// SIMATIC S7-200 project (STEP 7-Micro/WIN), CPU 224 REL 01.10

SYMBOL_TABLE IN/OUT
                 I0.0     // 水流量脉冲信号 0~3HZ,对应0~540M3/h
                 I0.1     // 变频器保护
                 I0.2     // 变频器输出控制权标定 脉冲转换 PLC/人操
                 I0.3     // 1#机变频电路 应答
                 I0.4     // 1#机系统电源电路 应答
                 I0.5     // 1#机变频电路 备妥
                 I0.6     // 1#机系统电源电路 备妥
                 I0.7     // 1#机电路热保护
                 I1.0     // 音响确认/试验
                 I1.1     // 2#机变频电路 应答
                 I1.2     // 2#机系统电源电路 应答
                 I1.3     // 2#机变频电路 备妥
                 I1.4     // 2#机系统电源电路 备妥
                 I1.5     // 2#机电路热保护
                 I2.0     // 3#机系统电源电路 应答
                 I2.1     // 3#机系统电源电路 备妥
                 I2.2     // 3#机电路热保护
                 I2.3     // 备用
                 Q0.0     // 1#机(电路)变频驱动
                 Q0.1     // 1#机系统电源驱动
                 Q0.2     // 2#机(电路)变频驱动
                 Q0.3     // 2#机系统电源驱动
                 Q0.4     // 停变频 复位自启动
                 Q0.5     // 1#操作提示
                 Q0.6     // 2#操作提示
                 Q0.7     // 共同部分操作提示
                 Q1.0     // 驱动报警音响
                 Q1.1     // 变频器输出由PLC控制 驱动指示灯
                 Q2.0     // 3#机系统电源驱动
                 Q2.1     // 备用
                 Q2.2     // 备用
                 Q2.3     // 备用
                 M0.0     // F1 1#机变频电路启动/停止
                 M0.1     // F2 1#机系统电源驱动的启动/停止
                 M0.2     // F3 2#机变频电路启动/停止
                 M0.3     // F4 2#机系统电源驱动的启动/停止
                 M0.4     // F5 3#机系统电源驱动的启动/停止
                 M0.5     // F6 变频手动输出设置调出
                 M0.6     // F7 待机/手动/自动切换
                 M0.7     // F8 赋值操作调出
                 AIW0     // 给水压力
                 AIW2     // 备用
                 AIW4     // 备用
                 AIW6     // 备用
                 AQW0     // 变频器输出频率控制
                 AQW2     // 备用
END_SYMBOL_TABLE

SYMBOL_TABLE OTHER
                 VD844    // Process Variable
                 VD848    // Loop Setpoint
                 VD852    // Calculated Loop Output
                 VD856    // Loop Gain
                 VD860    // Sample Time
                 VD864    // Integral Time
                 VD1012   // 供水安全值
                 VD1016   // 泵出口压力额定值
                 VD1020   // 泵供水量额定值
END_SYMBOL_TABLE

ORGANIZATION_BLOCK MAIN:OB1
TITLE= 
// 项目、设备信息
// 供水系统由2台55kw电机驱动的离心式水泵和1台30kw水泵组成工艺设备，其中55kw电机驱动的为主供水泵，额定压头420Kpa,额定流量250M3/h。正常供水量在额定流量范围内，一开一备。30kw电机驱动的为紧急泵，特殊工况下使用。系统设计为１台主供水泵由55kw变频器驱动，实现最佳节能控制，这台变频器还用于软启动两台水泵。（通过电气切换，在１台泵变频启动后，实行变频供电和系统电源切换，转由系统电源供电，变频器再去启动另１台泵。）在某些工况下，可能２台55kw泵同时运行。系统运行方式设计为"人操"和"ＰＬＣ"两种方式。
// 
// 系统注释
// 1、系统启动时，首先通过INIT子程序将系统运行模式置为待机状态，并初始化TD200显示屏参数。
// 2、系统中，两台55kW水泵分别由水泵1变频控制输出和水泵2变频控制输出控制，通过一台55kW变频器实现软启动和变频调速，以适应用水量变化。
// 3.、通过电气切换，在1#泵变频启动后，实行变频供电和系统电源切换，转由系统电源供电，变频器再去启动2#泵。
// 4、同时，30kW的水泵3控制输出在主泵异常时作为紧急备用，由F5键控制启停。
// 5.、小区物业管理人员可以通过TD200显示屏实时查看水泵状态、压力和流量数据。
// 6.、正常运行中，程序利用流量定时器计算每台水泵的流量，存储在流量计算结果中。
// 7、同时通过压力显示定时器定期更新压力数据到显示屏，确保物业人员随时掌握供水情况。
// 8、系统支持手动和自动两种模式切换，通过F7键触发，修改模式时确保水泵1变频控制输出已稳定，避免操作冲突。
// 9、在手动模式下，操作员可通过F1键启动1#机变频运行，但需变频器无故障且就绪时才会置位。
// 10、此外，F3键和F5键分别控制2#机和3#机的启停。
// 11、变频器的频率调整通过F6键实现，输出频率被严格限制在0-50Hz范围内，以保护设备不过载。
// 12、当切换至自动模式时，系统依靠PID调节自动控制水泵运行，维持恒定水压，此功能仅在自动模式下生效。
// 13、系统还会实时监控水泵1运行反馈等信号，并在TD200上显示状态。
// 14、安全性方面，若检测到水泵1热保护故障，程序立即复位水泵1变频控制输出和系统电源输出，并通过报警音响输出发出提示。
// 15、正常情况下，TD200显示屏显示PLC及1#机泵、2#机泵、3#机泵和变频器的运行状态，以及压力和流量测量值。
// 16、当有故障发生时，TD200显示屏显示汉字报警信息，PLC驱动音响报警，并自动停止故障设备。
// 17、操作人员可按确认键确认报警信息，按音响试验/消除按钮关闭音响，然后处理故障。
// 
// 
// 附加信息
// 正常情况下，TD200显示屏显示ＰＬＣ，１＃机泵，２＃机泵，３＃机泵和变频器的运行状态以及压力和流量测量值。当有故障发生时，TD200显示屏显示汉字的报警信息，同时ＰＬＣ驱动音响进行声音报警，ＰＬＣ自动停止发生故障的电气设备，以确保安全。操作人员可按确认键确认汉字的报警信息，按音响试验／消除按钮关闭音响，然后对故障进行处理。
// 
// 
BEGIN
Network 1 // 初始化
//  
// NETWORK COMMENTS
//  
// 
LD     SM0.1
CALL   INIT:SBR0
?000
Network 2 // 使能PID控制中断程序
// 
// 
LD     SM0.0
CALL   SBR_PID:SBR8
Network 3 // 流量脉冲计时
// 
// 
LD     SM0.0
TONR   T1, +32760
Network 4
LD     SM0.0
A      T1
MOVR   0.0, VD318
AENO
MOVR   0.0, VD338
AENO
MOVR   0.0, VD358
Network 5 // 显示压力
// 
// 
LD     SM0.0
AN     M3.1
TON    T103, +10
Network 6
// 
// 
LD     SM0.0
A      T103
CALL   P_DISPLAY:SBR1
=      M3.1
Network 7 // 显示电机与变频状态
// 
// 
LD     SM0.0
CALL   S_DISPLY:SBR2
Network 8
LD     SM0.0
AN     M2.1
R      M0.0, 5
Network 9 // F1键变频操作1#机
// 
// 
LD     SM0.0
A      M2.1
CALL   F1_CTRL1:SBR3
Network 10 // F2 1#机系统电源操作
// 
// 
LD     SM0.0
A      M2.1
CALL   F2_CTRL1:SBR4
Network 11 // F3键变频操作2#机
// 
// 
LD     SM0.0
A      M2.1
CALL   F3_CTRL2:SBR5
Network 12 // F4 2#机系统电源操作
// 
// 
LD     SM0.0
A      M2.1
CALL   F4_CTRL2:SBR6
Network 13 // F5 操3#机
// 
// 
LD     SM0.0
A      M2.1
CALL   F5_CTRL3:SBR7
Network 14 // 手动设置变频器输出
// 
// 
LD     SM0.0
A      M2.0
R      M0.5, 1
Network 15
LD     SM0.0
AN     M2.0
CALL   F6_FCMOUT:SBR9
Network 16 // 待机/手动/自动切换
// 
// 
LD     SM0.0
CALL   F7_SRMA:SBR10
Network 17 // 赋值操作
// 
// 
LD     SM0.0
CALL   F8_ASSIGN:SBR11
Network 18 // 故障
// 
// 
LD     SM0.0
CALL   E_FAULT:SBR16
Network 19 // 提示
// 
// 
LD     SM0.0
CALL   O_NOTE:SBR17
Network 20 // 报警
// 
// 
LD     SM0.0
CALL   ALARM:SBR18
END_ORGANIZATION_BLOCK

SUBROUTINE_BLOCK INIT:SBR0
TITLE= 
// SUBROUTINE COMMENTS
// Press F1 for help and example program
//  
BEGIN
Network 1 // 联接和使能中断程序
// 
// 
LD     SM0.0
MOVB   0, VB940
ATCH   Q_DISPLAY:INT0, 0
ENI
Network 2
LD     SM0.0
ATCH   FC_FAULT:INT1, 3
ENI
Network 3 // 设置初始状态为待机
// 
// 
LD     SM0.0
MOVB   0, MB2
Network 4 // 设置TD200初始显示
// 
// 
LD     SM0.1
MOVB   16#0, VB14
AENO
MOVB   16#2, VB15
AENO
MOVB   16#20, VB16
AENO
MOVW   16#0, VW17
AENO
MOVB   16#0, VB19
Network 5 // 首次扫描计算K,B
// 
// 
LD     SM0.0
MOVR   0.25, VD1060
AENO
*R     VD1020, VD1060
AENO
MOVR   0.4, VD1064
AENO
*R     VD1020, VD1064
AENO
MOVR   0.55, VD1068
*R     VD1020, VD1068
Network 6
LD     SM0.0
MOVR   0.7, VD1072
AENO
*R     VD1020, VD1072
AENO
MOVR   0.8, VD1076
AENO
*R     VD1020, VD1076
AENO
MOVR   0.9, VD1080
*R     VD1020, VD1080
Network 7
LD     SM0.0
MOVR   VD1020, VD1084
Network 8
LD     SM0.0
CALL   CO_FUCTION:SBR15, VD1024, VD1028, VD1056, VD1060, VD1088, VD1092
Network 9
LD     SM0.0
CALL   CO_FUCTION:SBR15, VD1028, VD1032, VD1060, VD1064, VD1096, VD1100
Network 10
LD     SM0.0
CALL   CO_FUCTION:SBR15, VD1032, VD1036, VD1064, VD1068, VD1104, VD1108
Network 11
LD     SM0.0
CALL   CO_FUCTION:SBR15, VD1036, VD1040, VD1068, VD1072, VD1112, VD1116
Network 12
LD     SM0.0
CALL   CO_FUCTION:SBR15, VD1040, VD1044, VD1072, VD1076, VD1120, VD1124
Network 13
LD     SM0.0
CALL   CO_FUCTION:SBR15, VD1044, VD1048, VD1076, VD1080, VD1128, VD1132
Network 14
LD     SM0.0
CALL   CO_FUCTION:SBR15, VD1048, VD1052, VD1080, VD1084, VD1136, VD1140
Network 15 // 设置变频器初始输出为50Hz
// 
// 
LD     SM0.0
MOVR   50.0, VD380
AENO
MOVR   VD380, VD852
/R     50.0, VD852
END_SUBROUTINE_BLOCK

SUBROUTINE_BLOCK P_DISPLAY:SBR1
TITLE= 
// SUBROUTINE COMMENTS
// Press F1 for help and example program
//  
BEGIN
Network 1
LD     SM0.0
LPS
XORW   VW948, VW948
MOVW   AIW0, VW950
A      V950.7
MOVW   16#FFFF, VW948
LPP
+D     -6400, VD948
AENO
DTR    VD948, VD948
Network 2
LD     SM0.0
LPS
/R     25600.0, VD948
AENO
*R     1200.0, VD948
AENO
MOVR   VD948, VD1000
LRD
ROUND  VD948, VD948
LPP
MOVW   VW950, VW312
AENO
MOVW   VW950, VW332
AENO
MOVW   VW950, VW352
END_SUBROUTINE_BLOCK

SUBROUTINE_BLOCK S_DISPLY:SBR2
TITLE= 
// SUBROUTINE COMMENTS
// Press F1 for help and example program
//  
BEGIN
Network 1 // 显示电机和变频状态
// 
// 
LD     SM0.0
MOVD   +100000, VD952
Network 2 // NETWORK TITLE (single line)
//  
// NETWORK COMMENTS
//  
// 
LD     SM0.0
A      I0.7
+D     +1, VD952
Network 3 // NETWORK TITLE (single line)
//  
// NETWORK COMMENTS
//  
// 
LD     SM0.0
A      I0.4
+D     +10, VD952
Network 4 // NETWORK TITLE (single line)
//  
// NETWORK COMMENTS
//  
// 
LD     SM0.0
A      I0.6
+D     +100, VD952
Network 5 // NETWORK TITLE (single line)
//  
// NETWORK COMMENTS
//  
// 
LD     SM0.0
A      I0.3
+D     +1000, VD952
Network 6 // NETWORK TITLE (single line)
//  
// NETWORK COMMENTS
//  
// 
LD     SM0.0
A      I0.5
+D     +10000, VD952
Network 7
LD     SM0.0
MOVD   VD952, VD386
AENO
MOVD   +200000, VD952
Network 8 // NETWORK TITLE (single line)
//  
// NETWORK COMMENTS
//  
// 
LD     SM0.0
A      I1.5
+D     +1, VD952
Network 9 // NETWORK TITLE (single line)
//  
// NETWORK COMMENTS
//  
// 
LD     SM0.0
A      I1.2
+D     +10, VD952
Network 10 // NETWORK TITLE (single line)
//  
// NETWORK COMMENTS
//  
// 
LD     SM0.0
A      I1.4
+D     +100, VD952
Network 11 // NETWORK TITLE (single line)
//  
// NETWORK COMMENTS
//  
// 
LD     SM0.0
A      I1.1
+D     +1000, VD952
Network 12 // NETWORK TITLE (single line)
//  
// NETWORK COMMENTS
//  
// 
LD     SM0.0
A      I1.3
+D     +10000, VD952
Network 13
LD     SM0.0
MOVD   VD952, VD392
AENO
MOVD   +400000, VD952
Network 14 // NETWORK TITLE (single line)
//  
// NETWORK COMMENTS
//  
// 
LD     SM0.0
A      I0.1
+D     +1, VD952
Network 15 // NETWORK TITLE (single line)
//  
// NETWORK COMMENTS
//  
// 
LD     SM0.0
A      Q1.1
+D     +10, VD952
Network 16 // NETWORK TITLE (single line)
//  
// NETWORK COMMENTS
//  
// 
LD     SM0.0
A      I2.2
+D     +100, VD952
Network 17 // NETWORK TITLE (single line)
//  
// NETWORK COMMENTS
//  
// 
LD     SM0.0
A      I2.0
+D     +1000, VD952
Network 18 // NETWORK TITLE (single line)
//  
// NETWORK COMMENTS
//  
// 
LD     SM0.0
A      I2.1
+D     +10000, VD952
Network 19
LD     SM0.0
MOVD   VD952, VD400
END_SUBROUTINE_BLOCK

SUBROUTINE_BLOCK F1_CTRL1:SBR3
TITLE= 
// SUBROUTINE COMMENTS
// Press F1 for help and example program
//  
BEGIN
Network 1
LD     SM0.0
LDB=   VB16, 16#20
AB=    VB15, 16#1
OB=    VB16, 16#A0
ALD
AB=    VB14, 0
AB=    VB17, 0
AB=    VB18, 0
AB=    VB19, 0
=      M1.0
Network 2 // 变频启动1#机
//  
// NETWORK COMMENTS
//  
// 
LDN    Q0.0
A      M0.0
LPS
A      M1.0
AN     Q0.1
LPS
AN     I0.7
S      V14.7, 1
LPP
A      I0.7
LPS
AN     I0.1
S      V14.4, 1
LPP
A      I0.1
LPS
AN     I0.5
S      V15.6, 1
LPP
A      I0.5
LPS
A      Q0.2
S      V15.5, 1
LPP
AN     Q0.2
S      V17.4, 1
S      V582.0, 1
MOVW   VW15, AC0
R      V15.0, 1
R      V16.5, 1
R      V16.7, 1
LPP
R      M0.0, 1
Network 3
LD     V17.4
TON    T37, +30
A      V582.1
S      Q0.0, 1
MOVW   AC0, VW15
R      V17.4, 1
R      V582.1, 1
Network 4
LDN    V582.1
A      T37
MOVW   AC0, VW15
R      V582.0, 1
R      V17.4, 1
Network 5 // 停1#机变频
// 
// 
LD     Q0.0
A      M0.0
LPS
A      M1.0
S      V17.3, 1
MOVW   VW15, AC0
R      V15.0, 1
R      V16.5, 1
R      V16.7, 1
S      V602.0, 1
LPP
R      M0.0, 1
Network 6
LD     V17.3
TON    T38, +30
A      V602.1
R      Q0.0, 1
MOVW   AC0, VW15
R      V17.3, 1
R      V602.1, 1
Network 7
LDN    V602.1
A      T38
MOVW   AC0, VW15
R      V602.0, 1
R      V17.3, 1
END_SUBROUTINE_BLOCK

SUBROUTINE_BLOCK F2_CTRL1:SBR4
TITLE= 
// SUBROUTINE COMMENTS
// Press F1 for help and example program
//  
BEGIN
Network 1 // 启1#机系统电源
//  
// NETWORK COMMENTS
//  
// 
LDN    Q0.1
A      M0.1
LPS
A      M1.0
LPS
AN     I0.6
S      V15.6, 1
LPP
A      I0.6
S      V17.2, 1
S      V622.0, 1
MOVW   VW15, AC0
R      V15.0, 1
R      V16.5, 1
R      V16.7, 1
LPP
R      M0.1, 1
Network 2
LD     Q0.0
TOF    T97, +400
Network 3
LD     V17.2
TON    T39, +30
A      V622.1
LPS
LD     Q0.0
ON     T97
ALD
S      V14.0, 1
S      M4.1, 1
S      M5.1, 1
LPP
LPS
AN     Q0.0
A      T97
S      Q0.1, 1
LRD
MOVW   AC0, VW15
LRD
R      V17.2, 1
LPP
R      V622.1, 1
Network 4
LDN    V622.1
A      T39
MOVW   AC0, VW15
R      V622.0, 1
R      V17.2, 1
Network 5 // 停1#机系统电源
// 
// 
LD     Q0.1
A      M0.1
LPS
A      M1.0
S      V17.0, 1
MOVW   VW15, AC0
R      V15.0, 1
R      V16.5, 1
R      V16.7, 1
S      V662.0, 1
LPP
R      M0.1, 1
Network 6
LD     V17.0
TON    T40, +30
A      V662.1
R      Q0.1, 1
MOVW   AC0, VW15
R      V17.0, 1
R      V662.1, 1
Network 7
LDN    V662.1
A      T40
MOVW   AC0, VW15
R      V662.0, 1
R      V17.0, 1
END_SUBROUTINE_BLOCK

SUBROUTINE_BLOCK F3_CTRL2:SBR5
TITLE= 
// SUBROUTINE COMMENTS
// Press F1 for help and example program
//  
BEGIN
Network 1 // 变频启动2#机
//  
// NETWORK COMMENTS
//  
// 
LDN    Q0.2
A      M0.2
LPS
A      M1.0
AN     Q0.3
LPS
AN     I1.5
S      V14.6, 1
LPP
A      I1.5
LPS
AN     I0.1
S      V14.4, 1
LPP
A      I0.1
LPS
AN     I1.3
S      V15.6, 1
LPP
A      I1.3
LPS
A      Q0.0
S      V15.5, 1
LPP
AN     Q0.0
S      V17.1, 1
S      V642.0, 1
MOVW   VW15, AC0
R      V15.0, 1
R      V16.5, 1
R      V16.7, 1
LPP
R      M0.2, 1
Network 2
LD     V17.1
TON    T41, +30
A      V642.1
S      Q0.2, 1
MOVW   AC0, VW15
R      V17.1, 1
R      V642.1, 1
Network 3
LDN    V642.1
A      T41
MOVW   AC0, VW15
R      V642.0, 1
R      V17.1, 1
Network 4 // 停2#机变频
// 
// 
LD     Q0.2
A      M0.2
LPS
A      M1.0
S      V16.4, 1
MOVW   VW15, AC0
R      V15.0, 1
R      V16.7, 1
R      V16.5, 1
S      V422.0, 1
LPP
R      M0.2, 1
Network 5
LD     V16.4
TON    T42, +30
A      V422.1
R      Q0.2, 1
MOVW   AC0, VW15
R      V16.4, 1
R      V422.1, 1
Network 6
LDN    V422.1
A      T42
MOVW   AC0, VW15
R      V422.0, 1
R      V16.4, 1
END_SUBROUTINE_BLOCK

SUBROUTINE_BLOCK F4_CTRL2:SBR6
TITLE= 
// SUBROUTINE COMMENTS
// Press F1 for help and example program
//  
BEGIN
Network 1 // 启2#机系统电源
//  
// NETWORK COMMENTS
//  
// 
LDN    Q0.3
A      M0.3
LPS
A      M1.0
LPS
AN     I1.4
S      V15.6, 1
LPP
A      I1.4
S      V16.3, 1
S      V442.0, 1
MOVW   VW15, AC0
R      V15.0, 1
R      V16.5, 1
R      V16.7, 1
LPP
R      M0.3, 1
Network 2
LD     Q0.2
TOF    T98, +400
Network 3
LD     V16.3
TON    T43, +30
A      V442.1
LPS
LD     Q0.2
ON     T98
ALD
S      V14.0, 1
S      M5.2, 1
S      M4.1, 1
LPP
LPS
AN     Q0.2
A      T98
S      Q0.3, 1
LRD
MOVW   AC0, VW15
LRD
R      V16.3, 1
LPP
R      V442.1, 1
Network 4
LDN    V442.1
A      T43
MOVW   AC0, VW15
R      V442.0, 1
R      V16.3, 1
Network 5 // 停2#机系统电源
// 
// 
LD     Q0.3
A      M0.3
LPS
A      M1.0
S      V16.2, 1
MOVW   VW15, AC0
R      V15.0, 1
R      V16.5, 1
R      V16.7, 1
S      V462.0, 1
LPP
R      M0.3, 1
Network 6
LD     V16.2
TON    T44, +30
A      V462.1
R      Q0.3, 1
MOVW   AC0, VW15
R      V16.2, 1
R      V462.1, 1
Network 7
LDN    V462.1
A      T44
MOVW   AC0, VW15
R      V462.0, 1
R      V16.2, 1
END_SUBROUTINE_BLOCK

SUBROUTINE_BLOCK F5_CTRL3:SBR7
TITLE= 
// SUBROUTINE COMMENTS
// Press F1 for help and example program
//  
BEGIN
Network 1 // 启动3#电机
// 
// 
LDN    Q2.0
A      M0.4
LPS
A      M1.0
LPS
AN     I2.2
S      V14.5, 1
LPP
A      I2.2
LPS
AN     I2.1
S      V15.6, 1
LPP
A      I2.1
S      V16.1, 1
S      V482.0, 1
MOVW   VW15, AC0
R      V15.0, 1
R      V16.5, 1
R      V16.7, 1
LPP
R      M0.4, 1
Network 2
LD     V16.1
TON    T45, +30
A      V482.1
S      Q2.0, 1
MOVW   AC0, VW15
R      V16.1, 1
R      V482.1, 1
Network 3
LDN    V482.1
A      T45
MOVW   AC0, VW15
R      V482.0, 1
R      V16.1, 1
Network 4 // 停3#机
// 
// 
LD     Q2.0
A      M0.4
LPS
A      M1.0
S      V16.0, 1
MOVW   VW15, AC0
R      V15.0, 1
R      V16.5, 1
R      V16.7, 1
S      V502.0, 1
LPP
R      M0.4, 1
Network 5
LD     V16.0
TON    T46, +30
A      V502.1
R      Q2.0, 1
MOVW   AC0, VW15
R      V16.0, 1
R      V502.1, 1
Network 6
LDN    V502.1
A      T46
MOVW   AC0, VW15
R      V502.0, 1
R      V16.0, 1
END_SUBROUTINE_BLOCK

SUBROUTINE_BLOCK SBR_PID:SBR8
TITLE=This POU was created by the PID formula of the S7-200 Instruction Wizard.
// This subroutine initializes the variables used by the PID control logic and starts the PID Interrupt "PID".  To enable this configuration within the program, use SM0.0 to call this Subroutine from the MAIN program block every scan cycle.  This code configures PID 0.  See DB1 for the PID loop variable table starting at VB844.  
BEGIN
Network 1 // Instruction Wizard PID (See Properties for more details).  
// PID Initialization and control.
// This subroutine initializes the variables used by the PID control logic and starts the PID Interrupt "PID".  
// routine. The PID interrupt routine is called cyclically based on the PID sample time. For
// a complete description of the PID instruction see the S7-200 System Manual.
// Note:
// When the PID is in manual mode the output should be controlled by writing a normalized value
// (0.00 to 1.00) to the PID Output instead of changing the output directly. This will automatically
// provide a bumpless transfer when the PID is returned to automatic mode.
// 
LDN    SM0.1
JMP    0
PID    VB844, 0
NOT
MOVW   +0, VW900             //initialize PID interrupt counter
MOVB   100, SMB34            //Load time for PID interrupt routine
ATCH   PID:INT2, 10          //Set up an interrupt to invoke PID execution
ENI
Network 2
LBL    0
Network 3
LD     M2.0
AN     M3.3
TON    T52, +3600
Network 4
LD     M2.0
A      T52
LPS
AR<=   VD358, 24.2
S      M3.2, 1
LPP
=      M3.3
Network 5
LD     M2.0
A      M3.2
TON    T53, +600
+R     0.2, VD852
AENO
MOVR   VD852, VD380
*R     50.0, VD380
Network 6
LD     M2.0
A      T53
R      M3.2, 1
END_SUBROUTINE_BLOCK

SUBROUTINE_BLOCK F6_FCMOUT:SBR9
TITLE= 
// SUBROUTINE COMMENTS
// Press F1 for help and example program
//  
BEGIN
Network 1
LD     SM0.0
AB=    VB16, 16#20
LDB=   VB15, 16#1
OB=    VB15, 16#2
ALD
AB=    VB14, 0
AB=    VB17, 0
AB=    VB18, 0
AB=    VB19, 0
=      M1.1
Network 2 // 手动设置变频器输出
//  
// NETWORK COMMENTS
//  
// 
LDN    M1.2
A      M0.5
LPS
A      M1.1
S      V16.6, 1
R      V16.5, 1
S      M1.2, 1
LPP
R      M0.5, 1
Network 3
LD     SM0.0
A      M1.2
TON    T47, +30
Network 4
LD     SM0.0
A      T47
S      V16.5, 1
R      V16.6, 1
R      M1.2, 1
Network 5
LD     M1.2
A      M0.5
S      V16.5, 1
R      V16.6, 1
R      M0.5, 1
R      M1.2, 1
Network 6
LD     SM0.0
A      V378.2
LPS
AR>=   VD380, 50.0
MOVR   50.0, VD380
LRD
AR<=   VD380, 0.0
MOVR   0.0, VD380
LRD
MOVR   VD380, AC0
AENO
MOVR   AC0, VD852
/R     50.0, VD852
LRD
S      V16.5, 1
LRD
R      V16.6, 1
LPP
R      V378.2, 1
END_SUBROUTINE_BLOCK

SUBROUTINE_BLOCK F7_SRMA:SBR10
TITLE= 
// SUBROUTINE COMMENTS
// Press F1 for help and example program
//  
BEGIN
Network 1
LD     SM0.0
LDB=   VB16, 16#20
AB=    VB15, 16#2
OB=    VB16, 16#A0
ALD
AB=    VB14, 0
AB=    VB17, 0
AB=    VB18, 0
AB=    VB19, 0
=      M1.3
Network 2
LD     SM0.0
AB=    VB16, 16#20
AB=    VB15, 16#1
AB=    VB14, 0
AB=    VB17, 0
AB=    VB18, 0
AB=    VB19, 0
=      M1.4
Network 3 // 切换到手动
// 
// 
LD     M0.6
A      M1.3
S      V17.7, 1
S      V522.0, 1
MOVW   VW15, AC0
R      V15.1, 1
R      V16.5, 1
R      V16.7, 1
Network 4
LD     V17.7
TON    T48, +30
A      V522.1
MOVB   16#2, MB2
S      V15.0, 1
S      V16.5, 1
R      V17.7, 1
R      V522.1, 1
Network 5
LD     V17.7
AN     V522.1
A      T48
MOVW   AC0, VW15
R      V522.0, 1
R      V17.7, 1
Network 6 // 切换到自动
// 
// 
LD     M0.6
LPS
A      M1.4
R      V15.0, 1
R      V16.5, 1
S      V542.0, 1
S      V17.6, 1
LPP
R      M0.6, 1
Network 7
LD     V17.6
TON    T49, +30
A      V542.1
S      V16.5, 1
S      V16.7, 1
MOVB   16#3, MB2
R      V17.6, 1
R      V542.1, 1
Network 8
LD     V17.6
AN     V542.1
A      T49
S      V15.0, 1
S      V16.5, 1
R      V542.0, 1
S      M1.5, 1
R      V17.6, 1
Network 9 // 切换到待机
// 
// 
LD     M1.5
TON    T50, +10
Network 10
LD     T50
A      M1.4
S      V17.5, 1
S      V562.0, 1
R      V16.5, 1
R      V15.0, 1
R      M1.5, 1
Network 11
LD     V17.5
TON    T51, +30
A      V562.1
S      V16.5, 1
S      V15.1, 1
MOVB   0, MB2
R      V17.5, 1
R      V562.1, 1
Network 12
LD     V17.5
AN     V562.1
A      T51
R      V562.0, 1
S      V15.0, 1
S      V16.5, 1
R      V17.5, 1
END_SUBROUTINE_BLOCK

SUBROUTINE_BLOCK F8_ASSIGN:SBR11
TITLE= 
// SUBROUTINE COMMENTS
// Press F1 for help and example program
//  
BEGIN
Network 1 // 赋值操作
//  
// NETWORK COMMENTS
//  
// 
LD     SM0.0
LD     M1.3
O      M1.4
ALD
=      M1.6
Network 2
LDN    M1.7
A      M0.7
LPS
A      M1.6
MOVW   VW15, AC0
R      V15.0, 2
R      V16.5, 1
R      V16.7, 1
MOVB   16#FF, VB18
S      M1.7, 1
LPP
R      M0.7, 1
Network 3
LD     SM0.0
A      M1.7
LD     M0.7
OB=    VB18, 0
ALD
S      V19.7, 1
MOVB   0, VB18
R      M0.7, 1
R      M1.7, 1
Network 4
LD     V19.7
A      V842.1
MOVW   AC0, VW15
CALL   SAVE_P:SBR14
R      V19.7, 1
R      V842.1, 1
Network 5 // 系数计算
// 
// 
LD     SM0.0
CALL   CO_CALCULATE:SBR12
END_SUBROUTINE_BLOCK

SUBROUTINE_BLOCK CO_CALCULATE:SBR12
TITLE= 
// SUBROUTINE COMMENTS
// Press F1 for help and example program
//  
BEGIN
Network 1 // 系数计算
//  
// NETWORK COMMENTS
//  
// 
LD     V678.2
LPS
AR>=   VD680, VD1012
AR<    VD680, VD700
LPS
MOVR   VD680, VD1024
AENO
CALL   CO_FUCTION:SBR15, VD1024, VD1028, VD1056, VD1060, VD1088, VD1092
LPP
NOT
MOVR   VD1024, VD680
LPP
R      V678.2, 1
Network 2
//  
// NETWORK COMMENTS
//  
// 
LD     V698.2
LPS
AR>    VD700, VD680
AR<    VD700, VD720
LPS
MOVR   VD700, VD1028
AENO
CALL   CO_FUCTION:SBR15, VD1024, VD1028, VD1056, VD1060, VD1088, VD1092
CALL   CO_FUCTION:SBR15, VD1028, VD1032, VD1060, VD1064, VD1096, VD1100
LPP
NOT
MOVR   VD1028, VD700
LPP
R      V698.2, 1
Network 3
//  
// NETWORK COMMENTS
//  
// 
LD     V718.2
LPS
AR>    VD720, VD700
AR<    VD720, VD740
LPS
MOVR   VD720, VD1032
AENO
CALL   CO_FUCTION:SBR15, VD1028, VD1032, VD1060, VD1064, VD1096, VD1100
CALL   CO_FUCTION:SBR15, VD1032, VD1036, VD1064, VD1068, VD1104, VD1108
LPP
NOT
MOVR   VD1032, VD720
LPP
R      V718.2, 1
Network 4
//  
// NETWORK COMMENTS
//  
// 
LD     V738.2
LPS
AR>    VD740, VD720
AR<    VD740, VD760
LPS
MOVR   VD740, VD1036
AENO
CALL   CO_FUCTION:SBR15, VD1032, VD1036, VD1064, VD1068, VD1104, VD1108
CALL   CO_FUCTION:SBR15, VD1036, VD1040, VD1068, VD1072, VD1112, VD1116
LPP
NOT
MOVR   VD1036, VD740
LPP
R      V738.2, 1
Network 5
//  
// NETWORK COMMENTS
//  
// 
LD     V758.2
LPS
AR>    VD760, VD740
AR<    VD760, VD780
LPS
MOVR   VD760, VD1040
AENO
CALL   CO_FUCTION:SBR15, VD1036, VD1040, VD1068, VD1072, VD1112, VD1116
CALL   CO_FUCTION:SBR15, VD1040, VD1044, VD1072, VD1076, VD1120, VD1124
LPP
NOT
MOVR   VD1040, VD760
LPP
R      V758.2, 1
Network 6
//  
// NETWORK COMMENTS
//  
// 
LD     V778.2
LPS
AR>    VD780, VD760
AR<    VD780, VD800
LPS
MOVR   VD780, VD1044
AENO
CALL   CO_FUCTION:SBR15, VD1040, VD1044, VD1072, VD1076, VD1120, VD1124
CALL   CO_FUCTION:SBR15, VD1044, VD1048, VD1076, VD1080, VD1128, VD1132
LPP
NOT
MOVR   VD1044, VD780
LPP
R      V778.2, 1
Network 7
//  
// NETWORK COMMENTS
//  
// 
LD     V798.2
LPS
AR>    VD800, VD780
AR<    VD800, VD820
LPS
MOVR   VD800, VD1048
AENO
CALL   CO_FUCTION:SBR15, VD1044, VD1048, VD1076, VD1080, VD1128, VD1132
CALL   CO_FUCTION:SBR15, VD1048, VD1052, VD1080, VD1084, VD1136, VD1140
LPP
NOT
MOVR   VD1048, VD800
LPP
R      V798.2, 1
Network 8
//  
// NETWORK COMMENTS
//  
// 
LD     V818.2
LPS
AR>    VD820, VD800
AR<=   VD820, VD1016
LPS
MOVR   VD820, VD1052
AENO
CALL   CO_FUCTION:SBR15, VD1048, VD1052, VD1080, VD1084, VD1136, VD1140
LPP
NOT
MOVR   VD1052, VD820
LPP
R      V818.2, 1
END_SUBROUTINE_BLOCK

SUBROUTINE_BLOCK SP_SET:SBR13
TITLE= 
// SUBROUTINE COMMENTS
// Press F1 for help and example program
//  
BEGIN
Network 1 // 计算设定值
// 
// 
LD     SM0.0
AR<    VD358, VD1060
MOVR   VD1088, AC1
AENO
*R     VD358, AC1
AENO
MOVR   AC1, VD956
+R     VD1092, VD956
Network 2
LD     SM0.0
AR>=   VD358, VD1060
AR<    VD358, VD1064
MOVR   VD1096, AC1
AENO
*R     VD358, AC1
AENO
MOVR   AC1, VD956
+R     VD1100, VD956
Network 3
LD     SM0.0
AR>=   VD358, VD1064
AR<    VD358, VD1068
MOVR   VD1104, AC1
AENO
*R     VD358, AC1
AENO
MOVR   AC1, VD956
+R     VD1108, VD956
Network 4
LD     SM0.0
AR>=   VD358, VD1068
AR<    VD358, VD1072
MOVR   VD1112, AC1
AENO
*R     VD358, AC1
AENO
MOVR   AC1, VD956
+R     VD1116, VD956
Network 5
LD     SM0.0
AR>=   VD358, VD1072
AR<    VD358, VD1076
MOVR   VD1120, AC1
AENO
*R     VD358, AC1
AENO
MOVR   AC1, VD956
+R     VD1124, VD956
Network 6
LD     SM0.0
AR>=   VD358, VD1076
AR<    VD358, VD1080
MOVR   VD1128, AC1
AENO
*R     VD358, AC1
AENO
MOVR   AC1, VD956
+R     VD1132, VD956
Network 7
LD     SM0.0
AR>=   VD358, VD1080
AR<    VD358, VD1084
MOVR   VD1136, AC1
AENO
*R     VD358, AC1
AENO
MOVR   AC1, VD956
+R     VD1140, VD956
Network 8
LD     SM0.0
AR>=   VD358, VD1084
MOVR   VD1052, VD956
Network 9
LD     SM0.0
MOVR   VD956, VD848
/R     1200.0, VD848
Network 10
LD     SM0.0
AR>=   1.0, VD848
NOT
MOVR   1.0, VD848
Network 11
LD     SM0.0
AR<=   0.0, VD848
NOT
MOVR   0.0, VD848
END_SUBROUTINE_BLOCK

SUBROUTINE_BLOCK SAVE_P:SBR14
TITLE= 
// SUBROUTINE COMMENTS
// Press F1 for help and example program
//  
BEGIN
Network 1 // 系数存储
//  
// NETWORK COMMENTS
//  
// 
LD     SM0.0
MOVW   +1024, SMW32
AENO
MOVB   16#83, SMB31
Network 2
//  
// NETWORK COMMENTS
//  
// 
LD     SM0.0
MOVW   +1028, SMW32
AENO
MOVB   16#83, SMB31
Network 3
//  
// NETWORK COMMENTS
//  
// 
LD     SM0.0
MOVW   +1032, SMW32
AENO
MOVB   16#83, SMB31
Network 4
//  
// NETWORK COMMENTS
//  
// 
LD     SM0.0
MOVW   +1036, SMW32
AENO
MOVB   16#83, SMB31
Network 5
//  
// NETWORK COMMENTS
//  
// 
LD     SM0.0
MOVW   +1040, SMW32
AENO
MOVB   16#83, SMB31
Network 6
//  
// NETWORK COMMENTS
//  
// 
LD     SM0.0
MOVW   +1044, SMW32
AENO
MOVB   16#83, SMB31
Network 7
//  
// NETWORK COMMENTS
//  
// 
LD     SM0.0
MOVW   +1048, SMW32
AENO
MOVB   16#83, SMB31
Network 8
//  
// NETWORK COMMENTS
//  
// 
LD     SM0.0
MOVW   +1052, SMW32
AENO
MOVB   16#83, SMB31
END_SUBROUTINE_BLOCK

SUBROUTINE_BLOCK CO_FUCTION:SBR15
TITLE=计算系数K,B的函数
VAR_INPUT
y1:REAL;	// LD0 
y2:REAL;	// LD4 
x1:REAL;	// LD8 
x2:REAL;	// LD12 
END_VAR
VAR_OUTPUT
k:REAL;	// LD16 
b:REAL;	// LD20 
END_VAR
VAR
m1:REAL;	// LD24 
m2:REAL;	// LD28 
END_VAR
BEGIN
Network 1 // 计算系数函数
//  
// NETWORK COMMENTS
//  
// 
LD     SM0.0
MOVR   #y2:LD4, #m1:LD24
AENO
-R     #y1:LD0, #m1:LD24
AENO
MOVR   #x2:LD12, #m2:LD28
-R     #x1:LD8, #m2:LD28
Network 2
LD     SM0.0
MOVR   #m1:LD24, #k:LD16
AENO
/R     #m2:LD28, #k:LD16
AENO
MOVR   #x1:LD8, #m1:LD24
AENO
*R     #k:LD16, #m1:LD24
AENO
MOVR   #y1:LD0, #b:LD20
-R     #m1:LD24, #b:LD20
END_SUBROUTINE_BLOCK

SUBROUTINE_BLOCK E_FAULT:SBR16
TITLE= 
// SUBROUTINE COMMENTS
// Press F1 for help and example program
//  
BEGIN
Network 1 // 1#机热保护故障
// 
// 
LD     SM0.0
A      I0.7
ED
S      M4.0, 1
S      V14.7, 1
R      Q0.0, 2
Network 2 // 2#机热保护故障
// 
// 
LD     SM0.0
A      I1.5
ED
S      M4.0, 1
S      V14.6, 1
R      Q0.2, 2
Network 3 // 3#机热保护故障
// 
// 
LD     SM0.0
A      I2.2
ED
S      M4.0, 1
S      V14.5, 1
R      Q2.0, 1
Network 4 // 变频复位自启动
// 
// 
LD     SM0.0
A      Q0.4
TON    T54, +30
Network 5
LD     SM0.0
A      T54
R      Q0.4, 1
Network 6 // 变频器故障
// 
// 
LD     SM0.0
A      M3.0
AN     I0.1
TON    T55, +40
Network 7
LD     SM0.0
A      T55
EU
S      M4.0, 1
S      V14.4, 1
R      M3.0, 1
Network 8
LD     SM0.0
A      I0.1
EU
R      M3.0, 1
Network 9 // 1#机变频电路输出与反馈不一致
// 
// 
LD     SM0.0
A      Q0.0
TON    T56, +30
TOF    T57, +30
Network 10
LD     SM0.0
LD     T56
AN     I0.3
LDN    T57
A      I0.3
OLD
ALD
EU
S      M4.0, 1
R      Q0.0, 1
S      V14.3, 1
Network 11 // 1#机系统电源电路输出与反馈不一致
// 
// 
LD     SM0.0
A      Q0.1
TON    T58, +30
TOF    T59, +30
Network 12
LD     SM0.0
LD     T58
AN     I0.4
LDN    T59
A      I0.4
OLD
ALD
EU
S      M4.0, 1
R      Q0.1, 1
S      V14.3, 1
Network 13 // 2#机变频电路输出与反馈不一致
// 
// 
LD     SM0.0
A      Q0.2
TON    T60, +30
TOF    T61, +30
Network 14
LD     SM0.0
LD     T60
AN     I1.1
LDN    T61
A      I1.1
OLD
ALD
EU
S      M4.0, 1
R      Q0.2, 1
S      V14.2, 1
Network 15 // 2#机系统电源电路输出与反馈不一致
// 
// 
LD     SM0.0
A      Q0.3
TON    T62, +30
TOF    T63, +30
Network 16
LD     SM0.0
LD     T62
AN     I1.2
LDN    T63
A      I1.2
OLD
ALD
EU
S      M4.0, 1
R      Q0.3, 1
S      V14.2, 1
Network 17 // 3#机变频电路输出与反馈不一致
// 
// 
LD     SM0.0
A      Q2.0
TON    T101, +30
TOF    T102, +30
Network 18
LD     SM0.0
LD     T101
AN     I2.0
LDN    T102
A      I2.0
OLD
ALD
EU
S      M4.0, 1
R      Q2.0, 1
S      V14.1, 1
END_SUBROUTINE_BLOCK

SUBROUTINE_BLOCK O_NOTE:SBR17
TITLE= 
// SUBROUTINE COMMENTS
// Press F1 for help and example program
//  
BEGIN
Network 1 // 变频器输出控制权转换
//  
// NETWORK COMMENTS
//  
// 
LD     SM0.0
A      I0.2
ED
S      V15.7, 1
Network 2
LD     SM0.0
A      I0.2
ED
LPS
AN     Q1.1
S      Q1.1, 1
LPP
A      Q1.1
R      Q1.1, 1
Network 3
LD     SM0.0
A      Q1.1
ED
S      M4.1, 1
Network 4 // 启动备用机
// 
// 
LD     SM0.0
AN     I2.0
AR>=   VD318, VD1080
LPS
A      I0.3
AN     I1.2
AN     I1.1
TON    T104, +600
LPP
A      I1.1
AN     I0.4
AN     I0.3
TON    T105, +600
Network 5
LD     SM0.0
LD     T104
O      T105
ALD
EU
S      V15.4, 1
S      M4.1, 1
Network 6
LD     SM0.0
A      T104
=      M4.3
Network 7
LD     SM0.0
A      T105
=      M4.6
Network 8 // 停一台机
// 
// 
LD     SM0.0
AR<=   VD318, 229.9
LPS
A      I0.3
LD     I1.2
O      I2.0
ALD
TON    T106, +600
LPP
A      I1.1
LD     I0.4
O      I2.0
ALD
TON    T107, +600
Network 9
LD     SM0.0
LD     T106
O      T107
ALD
EU
S      V15.3, 1
S      M4.1, 1
Network 10
LD     SM0.0
A      T106
=      M4.4
Network 11
LD     SM0.0
A      T107
=      M4.7
Network 12 // 操作阀门
// 
// 
LD     SM0.0
LD     I0.3
O      I1.1
O      I2.0
ALD
EU
S      V15.2, 1
S      M4.1, 1
Network 13
LD     SM0.0
LD     I0.4
O      I1.2
O      I2.0
ALD
ED
S      V15.2, 1
S      M4.1, 1
Network 14
LD     SM0.0
A      I0.3
ED
S      M3.4, 1
Network 15
LD     SM0.0
A      I1.1
ED
S      M3.5, 1
Network 16
LD     SM0.0
A      M3.4
TON    T108, +50
Network 17
LD     SM0.0
A      M3.5
TON    T109, +50
Network 18
LD     SM0.0
A      T108
LPS
AN     I0.4
S      V15.2, 1
S      M4.1, 1
LPP
R      M3.4, 1
Network 19
LD     SM0.0
A      T109
LPS
AN     I1.2
S      V15.2, 1
S      M4.1, 1
LPP
R      M3.5, 1
Network 20 // 1#机变频电路与变频输出控权不一致
// 
// 
LD     SM0.0
LD     Q1.1
AN     I0.5
LD     I0.5
AN     Q1.1
OLD
ALD
=      M4.2
EU
S      M4.1, 1
R      Q0.0, 1
Network 21 // 2#机变频电路与变频输出控权不一致
// 
// 
LD     SM0.0
LD     Q1.1
AN     I1.3
LD     I1.3
AN     Q1.1
OLD
ALD
=      M4.5
EU
S      M4.1, 1
R      Q0.2, 1
Network 22 // 压力,流量值不正常
// 
// 
LD     SM0.0
LD     I0.3
O      I0.4
O      I1.1
O      I1.2
O      I2.0
ALD
LDR<=  VD1000, VD1012
LDR>=  VD1000, VD1012
AR<    VD318, 48.4
OLD
OR>=   VD318, VD1020
ALD
=      M5.0
EU
S      M4.1, 1
Network 23 // 系统电源启动不安全确认
// 
// 
LD     V182.1
R      M5.1, 2
R      V182.1, 1
END_SUBROUTINE_BLOCK

SUBROUTINE_BLOCK ALARM:SBR18
TITLE= 
// SUBROUTINE COMMENTS
// Press F1 for help and example program
//  
BEGIN
Network 1 // 设置输出脉冲
//  
// NETWORK COMMENTS
//  
// 
LD     SM0.0
AN     M3.6
TON    T110, +20
Network 2
LD     SM0.0
A      M3.6
TON    T111, +20
Network 3
LD     SM0.0
A      T110
S      M3.6, 1
Network 4
LD     SM0.0
A      T111
R      M3.6, 1
Network 5
LD     SM0.0
AN     M3.7
TON    T112, +30
Network 6
LD     SM0.0
A      M3.7
TON    T113, +10
Network 7
LD     SM0.0
A      T112
S      M3.7, 1
Network 8
LD     SM0.0
A      T113
R      M3.7, 1
Network 9 // 音响报警
// 
// 
LD     SM0.0
A      M4.0
LPS
AN     M3.7
=      Q1.0
LPP
JMP    0
Network 10
LD     SM0.0
LD     M4.1
O      M6.0
ALD
A      M3.7
=      Q1.0
Network 11
LBL    0
Network 12
LD     SM0.0
A      I1.0
EU
LPS
AN     V960.0
S      M6.0, 1
LPP
A      V960.0
R      M6.0, 1
Network 13
LD     SM0.0
A      I1.0
EU
INCB   VB960
Network 14
LD     SM0.0
A      M4.1
EU
AN     M6.0
AN     M4.0
INCB   VB960
Network 15
LD     SM0.0
A      M4.0
EU
AN     M6.0
AN     M4.1
INCB   VB960
Network 16
LD     SM0.0
AB>=   VB960, 2
MOVB   0, VB960
Network 17
LD     SM0.0
A      I1.0
R      M4.0, 2
Network 18 // 1#机状态指示
//  
// NETWORK COMMENTS
//  
// 
LD     SM0.0
A      M4.4
LPS
AN     M3.7
=      Q0.5
LPP
JMP    1
Network 19
//  
// NETWORK COMMENTS
//  
// 
LD     SM0.0
A      M4.3
LPS
A      M3.7
=      Q0.5
LPP
JMP    1
Network 20
//  
// NETWORK COMMENTS
//  
// 
LD     SM0.0
A      M4.2
A      M3.6
=      Q0.5
Network 21
LBL    1
Network 22 // 2#机状态指示
//  
// NETWORK COMMENTS
//  
// 
LD     SM0.0
A      M4.7
LPS
AN     M3.7
=      Q0.6
LPP
JMP    2
Network 23
//  
// NETWORK COMMENTS
//  
// 
LD     SM0.0
A      M4.6
LPS
A      M3.7
=      Q0.6
LPP
JMP    2
Network 24
//  
// NETWORK COMMENTS
//  
// 
LD     SM0.0
A      M4.5
A      M3.6
=      Q0.6
Network 25
LBL    2
Network 26 // 共同部分指示
//  
// NETWORK COMMENTS
//  
// 
LD     SM0.0
A      M5.2
LPS
AN     M3.7
=      Q0.7
LPP
JMP    3
Network 27
//  
// NETWORK COMMENTS
//  
// 
LD     SM0.0
A      M5.1
LPS
A      M3.7
=      Q0.7
LPP
JMP    3
Network 28
//  
// NETWORK COMMENTS
//  
// 
LD     SM0.0
A      M5.0
A      M3.6
=      Q0.7
Network 29
LBL    3
END_SUBROUTINE_BLOCK

INTERRUPT_BLOCK Q_DISPLAY:INT0
TITLE=流量计算中断程序
BEGIN
Network 1
LD     SM0.0
INCB   VB940
AB>=   VB940, 2
LPS
MOVB   0, VB940
XORW   VW944, VW944
MOVW   T1, VW946
AENO
R      T1, 1
LRD
DTR    VD944, VD944
LPP
MOVR   36000.0, VD318
AENO
/R     VD944, VD318
AENO
MOVR   VD318, VD338
AENO
MOVR   VD318, VD358
END_INTERRUPT_BLOCK

INTERRUPT_BLOCK FC_FAULT:INT1
TITLE=变频器故障处理中断程序
BEGIN
Network 1 // 变频器故障中断
//  
// NETWORK COMMENTS
//  
// 
LD     SM0.0
S      Q0.4, 1
S      M3.0, 1
END_INTERRUPT_BLOCK

INTERRUPT_BLOCK PID:INT2
TITLE=This POU was created by the PID formula of the S7-200 Instruction Wizard.
// This interrupt routine implements Timed Interrupt for PID execution. This interrupt routine was attached in subroutine "SBR_PID".
BEGIN
Network 1 // Instruction Wizard PID (See Properties for more details).  
// Increment number of times routine is called
// 
LD     SM0.0
INCW   VW900
Network 2
LDW>=  VW900, VW1004         //Check if time to do PID calculation
MOVW   +0, VW900             //if so, clear the counter and continue
NOT
JMP    0                     //otherwise, jump to the end of the interrupt routine
Network 3 // Compute the normalized value and load it into the PID PV location
LD     SM0.0                 //Always
LPS                          //Clear the working area.
XORW   VW914, VW914          //read the analog value
MOVW   AIW0, VW916
A      V916.7                //Check the sign bit.
MOVW   16#FFFF, VW914        //Extend the sign.
LRD
+D     -6400, VD914          //Adjust for offset
LRD                          //and convert it to a real number and load it in the PV
DTR    VD914, VD844          //Normalize to a value between 0.0 and 1.0
LPP
/R     25600.0, VD844
Network 4
LD     SM0.0
CALL   SP_SET:SBR13
Network 5 // Clamp the value to a maximum of 1.0.
LDR>=  1.0, VD844
NOT
MOVR   1.0, VD844
Network 6 // Clamp the value to a minimum of 0.0.
LDR<=  0.0, VD844
NOT
MOVR   0.0, VD844
Network 7 // Perform PID calculation
LD     SM0.0                 //Always
A      M3.2                  //then perform PID calculation
A      M2.0
PID    VB844, 0
MOVR   VD852, VD380
*R     50.0, VD380
Network 8 // Scale the PID output and transfer it to the analog output
LD     SM0.0                 //Always
MOVR   VD852, VD914          //load the PID output to workspace
*R     25600.0, VD914        //scale the value
TRUNC  VD914, VD914          //convert the value to an integer
+D     +6400, VD914          //Adjust for offset
MOVW   VW916, AQW0           //and transfer it to the analog output
Network 9
LBL    0
END_INTERRUPT_BLOCK

DATA_BLOCK_TAB USER1
BEGIN
//DATA BLOCK COMMENTS
//Press F1 for help and example data block
//BEGIN TD200_BLOCK 0
// 
//(Comments within this block should not be edited or removed)
// 
VB0      'TD'
VB2      16#60               //Set Language to Chinese, set Update to as fast as possible 
VB3      16#F0               //Set the display to 20 character mode; Up key V3.2; Down key V3.3;
VB4      41                  //Set the number of messages
VB5      0                   //Set the Function Keys notification bits to M0.0 - M0.7
VW6      24                  //Set the starting address for messages to  VW24
VW8      14                  //Set the starting address for message enable bits to VW14
VW10     8888                //Global Password (if enabled)
VW12     256                 //Character Set = Simplified Chinese
//MESSAGE 1
//Message Enable Bit V14.7 
VB24     '1#机泵故障 !!!    '
VB42     16#1                //No Edit;Acknowledgement Notification V42.1; No Password;
VB43     16#0                //No Data; 0 Digits to the right of the decimal;
//MESSAGE 2
//Message Enable Bit V14.6 
VB44     '2#机泵故障!!!     '
VB62     16#1                //No Edit;Acknowledgement Notification V62.1; No Password;
VB63     16#0                //No Data; 0 Digits to the right of the decimal;
//MESSAGE 3
//Message Enable Bit V14.5 
VB64     '3#机泵故障!!!     '
VB82     16#1                //No Edit;Acknowledgement Notification V82.1; No Password;
VB83     16#0                //No Data; 0 Digits to the right of the decimal;
//MESSAGE 4
//Message Enable Bit V14.4 
VB84     '变频器故障!!!     '
VB102    16#1                //No Edit;Acknowledgement Notification V102.1; No Password;
VB103    16#0                //No Data; 0 Digits to the right of the decimal;
//MESSAGE 5
//Message Enable Bit V14.3 
VB104    '1#操作与反馈不一致'
VB122    16#1                //No Edit;Acknowledgement Notification V122.1; No Password;
VB123    16#0                //No Data; 0 Digits to the right of the decimal;
//MESSAGE 6
//Message Enable Bit V14.2 
VB124    '2#操作与反馈不一致'
VB142    16#1                //No Edit;Acknowledgement Notification V142.1; No Password;
VB143    16#0                //No Data; 0 Digits to the right of the decimal;
//MESSAGE 7
//Message Enable Bit V14.1 
VB144    '3#操作与反馈不一致'
VB162    16#1                //No Edit;Acknowledgement Notification V162.1; No Password;
VB163    16#0                //No Data; 0 Digits to the right of the decimal;
//MESSAGE 8
//Message Enable Bit V14.0 
VB164    '系统电源启动不安全'
VB182    16#1                //No Edit;Acknowledgement Notification V182.1; No Password;
VB183    16#0                //No Data; 0 Digits to the right of the decimal;
//MESSAGE 9
//Message Enable Bit V15.7 
VB184    '变频器输出控权转换'
VB202    16#1                //No Edit;Acknowledgement Notification V202.1; No Password;
VB203    16#0                //No Data; 0 Digits to the right of the decimal;
//MESSAGE 10
//Message Enable Bit V15.6 
VB204    '电路控权不在PLC   '
VB222    16#1                //No Edit;Acknowledgement Notification V222.1; No Password;
VB223    16#0                //No Data; 0 Digits to the right of the decimal;
//MESSAGE 11
//Message Enable Bit V15.5 
VB224    '变频正由另台机使用'
VB242    16#1                //No Edit;Acknowledgement Notification V242.1; No Password;
VB243    16#0                //No Data; 0 Digits to the right of the decimal;
//MESSAGE 12
//Message Enable Bit V15.4 
VB244    '启动备用机或3#机泵'
VB262    16#1                //No Edit;Acknowledgement Notification V262.1; No Password;
VB263    16#0                //No Data; 0 Digits to the right of the decimal;
//MESSAGE 13
//Message Enable Bit V15.3 
VB264    '停止一台机泵      '
VB282    16#1                //No Edit;Acknowledgement Notification V282.1; No Password;
VB283    16#0                //No Data; 0 Digits to the right of the decimal;
//MESSAGE 14
//Message Enable Bit V15.2 
VB284    '请操作泵出口阀门  '
VB302    16#1                //No Edit;Acknowledgement Notification V302.1; No Password;
VB303    16#0                //No Data; 0 Digits to the right of the decimal;
//MESSAGE 15
//Message Enable Bit V15.1 
VB304    '待机P:'
VB310    16#0                //No Edit;No Acknowledgement;No Password;
VB311    16#10               //Signed Word; 0 Digits to the right of the decimal;
VW312    16#0                //Embedded Data Value: Move data for display here.
VB314    'Q:'
VB316    16#0                //No Edit;No Acknowledgement;No Password;
VB317    16#51               //Real Double Word; 1 Digits to the right of the decimal;
VD318    16#0                //Embedded Data Value: Move data for display here.
VB322    '  '
//MESSAGE 16
//Message Enable Bit V15.0 
VB324    '手动P:'
VB330    16#0                //No Edit;No Acknowledgement;No Password;
VB331    16#10               //Signed Word; 0 Digits to the right of the decimal;
VW332    16#0                //Embedded Data Value: Move data for display here.
VB334    'Q:'
VB336    16#0                //No Edit;No Acknowledgement;No Password;
VB337    16#51               //Real Double Word; 1 Digits to the right of the decimal;
VD338    16#0                //Embedded Data Value: Move data for display here.
VB342    '  '
//MESSAGE 17
//Message Enable Bit V16.7 
VB344    '自动P:'
VB350    16#0                //No Edit;No Acknowledgement;No Password;
VB351    16#10               //Signed Word; 0 Digits to the right of the decimal;
VW352    16#0                //Embedded Data Value: Move data for display here.
VB354    'Q:'
VB356    16#0                //No Edit;No Acknowledgement;No Password;
VB357    16#51               //Real Double Word; 1 Digits to the right of the decimal;
VD358    16#0                //Embedded Data Value: Move data for display here.
VB362    '  '
//MESSAGE 18
//Message Enable Bit V16.6 
VB364    '变频输出设定Y:'
VB378    16#10               //Edit Notification V378.2; No Acknowledgement;No Password;
VB379    16#51               //Real Double Word; 1 Digits to the right of the decimal;
VD380    16#0                //Embedded Data Value: Move data for display here.
//MESSAGE 19
//Message Enable Bit V16.5 
VB384    16#0                //No Edit;No Acknowledgement;No Password;
VB385    16#40               //Unsigned Double Word; 0 Digits to the right of the decimal;
VD386    16#0                //Embedded Data Value: Move data for display here.
VB390    16#0                //No Edit;No Acknowledgement;No Password;
VB391    16#40               //Unsigned Double Word; 0 Digits to the right of the decimal;
VD392    16#0                //Embedded Data Value: Move data for display here.
VB396    '3&'
VB398    16#0                //No Edit;No Acknowledgement;No Password;
VB399    16#40               //Unsigned Double Word; 0 Digits to the right of the decimal;
VD400    16#0                //Embedded Data Value: Move data for display here.
//MESSAGE 20
//Message Enable Bit V16.4 
VB404    '断2#机变频电路确认'
VB422    16#1                //No Edit;Acknowledgement Notification V422.1; No Password;
VB423    16#0                //No Data; 0 Digits to the right of the decimal;
//MESSAGE 21
//Message Enable Bit V16.3 
VB424    '切换2#机电源确认  '
VB442    16#1                //No Edit;Acknowledgement Notification V442.1; No Password;
VB443    16#0                //No Data; 0 Digits to the right of the decimal;
//MESSAGE 22
//Message Enable Bit V16.2 
VB444    '断2#机系统电源确认'
VB462    16#1                //No Edit;Acknowledgement Notification V462.1; No Password;
VB463    16#0                //No Data; 0 Digits to the right of the decimal;
//MESSAGE 23
//Message Enable Bit V16.1 
VB464    '启动3#机紧急泵确认'
VB482    16#1                //No Edit;Acknowledgement Notification V482.1; No Password;
VB483    16#0                //No Data; 0 Digits to the right of the decimal;
//MESSAGE 24
//Message Enable Bit V16.0 
VB484    '停止3#机紧急泵确认'
VB502    16#1                //No Edit;Acknowledgement Notification V502.1; No Password;
VB503    16#0                //No Data; 0 Digits to the right of the decimal;
//MESSAGE 25
//Message Enable Bit V17.7 
VB504    '切换到手动确认    '
VB522    16#1                //No Edit;Acknowledgement Notification V522.1; No Password;
VB523    16#0                //No Data; 0 Digits to the right of the decimal;
//MESSAGE 26
//Message Enable Bit V17.6 
VB524    '切换到自动确认    '
VB542    16#1                //No Edit;Acknowledgement Notification V542.1; No Password;
VB543    16#0                //No Data; 0 Digits to the right of the decimal;
//MESSAGE 27
//Message Enable Bit V17.5 
VB544    '切换到待机确认    '
VB562    16#1                //No Edit;Acknowledgement Notification V562.1; No Password;
VB563    16#0                //No Data; 0 Digits to the right of the decimal;
//MESSAGE 28
//Message Enable Bit V17.4 
VB564    '变频软启动1#机确认'
VB582    16#1                //No Edit;Acknowledgement Notification V582.1; No Password;
VB583    16#0                //No Data; 0 Digits to the right of the decimal;
//MESSAGE 29
//Message Enable Bit V17.3 
VB584    '断1#机变频电路确认'
VB602    16#1                //No Edit;Acknowledgement Notification V602.1; No Password;
VB603    16#0                //No Data; 0 Digits to the right of the decimal;
//MESSAGE 30
//Message Enable Bit V17.2 
VB604    '切换1#机电源确认  '
VB622    16#1                //No Edit;Acknowledgement Notification V622.1; No Password;
VB623    16#0                //No Data; 0 Digits to the right of the decimal;
//MESSAGE 31
//Message Enable Bit V17.1 
VB624    '变频软启动2#机确认'
VB642    16#1                //No Edit;Acknowledgement Notification V642.1; No Password;
VB643    16#0                //No Data; 0 Digits to the right of the decimal;
//MESSAGE 32
//Message Enable Bit V17.0 
VB644    '断1#机系统电源确认'
VB662    16#1                //No Edit;Acknowledgement Notification V662.1; No Password;
VB663    16#0                //No Data; 0 Digits to the right of the decimal;
//MESSAGE 33
//Message Enable Bit V18.7 
VB664    '赋值Q=0.00QeP='
VB678    16#10               //Edit Notification V678.2; No Acknowledgement;No Password;
VB679    16#50               //Real Double Word; 0 Digits to the right of the decimal;
VD680    16#0                //Embedded Data Value: Move data for display here.
//MESSAGE 34
//Message Enable Bit V18.6 
VB684    '赋值Q=0.25QeP='
VB698    16#10               //Edit Notification V698.2; No Acknowledgement;No Password;
VB699    16#50               //Real Double Word; 0 Digits to the right of the decimal;
VD700    16#0                //Embedded Data Value: Move data for display here.
//MESSAGE 35
//Message Enable Bit V18.5 
VB704    '赋值Q=0.40QeP='
VB718    16#10               //Edit Notification V718.2; No Acknowledgement;No Password;
VB719    16#50               //Real Double Word; 0 Digits to the right of the decimal;
VD720    16#0                //Embedded Data Value: Move data for display here.
//MESSAGE 36
//Message Enable Bit V18.4 
VB724    '赋值Q=0.55QeP='
VB738    16#10               //Edit Notification V738.2; No Acknowledgement;No Password;
VB739    16#50               //Real Double Word; 0 Digits to the right of the decimal;
VD740    16#0                //Embedded Data Value: Move data for display here.
//MESSAGE 37
//Message Enable Bit V18.3 
VB744    '赋值Q=0.70QeP='
VB758    16#10               //Edit Notification V758.2; No Acknowledgement;No Password;
VB759    16#50               //Real Double Word; 0 Digits to the right of the decimal;
VD760    16#0                //Embedded Data Value: Move data for display here.
//MESSAGE 38
//Message Enable Bit V18.2 
VB764    '赋值Q=0.80QeP='
VB778    16#10               //Edit Notification V778.2; No Acknowledgement;No Password;
VB779    16#50               //Real Double Word; 0 Digits to the right of the decimal;
VD780    16#0                //Embedded Data Value: Move data for display here.
//MESSAGE 39
//Message Enable Bit V18.1 
VB784    '赋值Q=0.90QeP='
VB798    16#10               //Edit Notification V798.2; No Acknowledgement;No Password;
VB799    16#50               //Real Double Word; 0 Digits to the right of the decimal;
VD800    16#0                //Embedded Data Value: Move data for display here.
//MESSAGE 40
//Message Enable Bit V18.0 
VB804    '赋值Q=1.00QeP='
VB818    16#10               //Edit Notification V818.2; No Acknowledgement;No Password;
VB819    16#50               //Real Double Word; 0 Digits to the right of the decimal;
VD820    16#0                //Embedded Data Value: Move data for display here.
//MESSAGE 41
//Message Enable Bit V19.7 
VB824    '赋值结束确认      '
VB842    16#1                //No Edit;Acknowledgement Notification V842.1; No Password;
VB843    16#0                //No Data; 0 Digits to the right of the decimal;
//END TD200_BLOCK 0
// 
//The following were generated by the S7-200 Instruction Wizard, PID Formula.  
//Parameter Table for PID 0.
// 
VD844    0.0                 //Process Variable
VD848    0.0                 //Loop Setpoint
VD852    0.0                 //Calculated Loop Output
VD856    1.2                 //Loop Gain
VD860    10.0                //Sample Time
VD864    10.0                //Integral Time
VD868    0.0                 //Derivative Time
VD872    0.0                 //Integral Sum or Bias
VD876    0.0                 //Value of Process Variable stored from last execution.
VW1004   30                  //PID运算周期
VD1012   210.0               //Pa 供水安全值
VD1016   420.0               //Pe 泵出口压力额定值
VD1020   242.0               //Qe 泵供水量额定值
VD1024   210.0               //P0
VD1028   262.5               //p1
VD1032   294.0               //p2
VD1036   325.5               //p3
VD1040   357.0               //p4
VD1044   378.0               //p5
VD1048   399.0               //p6
VD1052   420.0               //p7
VD1056   0.0                 //Q0
VD1060   60.5                //Q1
VD1064   96.8                //Q2
VD1068   133.1               //Q3
VD1072   169.4               //Q4
VD1076   193.6               //Q5
VD1080   217.8               //Q6
VD1084   242.0               //Q7
END_DATA_BLOCK_TAB
